(* Basic GVL for autodocs tests. *)
VAR_GLOBAL
    bSystemReady : BOOL;
    nCounter     : INT := 0;
END_VAR
VAR_GLOBAL CONSTANT
    cMaxCount : INT := 100;
END_VAR

(* stored: Version 1.1.0.1
   GVL GVL_Basic: Id {66666666-6666-6666-6666-666666666601} *)
